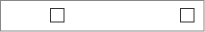
VISUALIZATION VISU_ConfigBOOLEntry  // 205x32
VAR_IN_OUT
    active : BOOL;
    editable : BOOL;
END_VAR
    Checkbox (48,0 45x30), variable: active, input disabled if: TRUE
    Checkbox (178,0 25x30), variable: editable
END_VISUALIZATION

(* stored: Version 1.1.0.1, ProductVersion 3.1.0.36
   Visu VISU_ConfigBOOLEntry: Id {a175e75a-f72f-48c3-bf55-1ce4a4306413} *)
